Staubli VAL3: refreshImport.pgx

program refreshImport(bool x_bShowLine (dimensions=1), string& x_sPath[] (dimensions=1))
  local num l_nLocal
  local string l_sEmpty
  local string l_sItem
begin
  //
  call use2:setSizeList(0,0,17,11)
  call use2:listcreate("USB")
  call use:stringCopy(l_sEmpty,sImport)
  call use2:listempty()
  //
  // build the list
  if libList(x_sPath[1],sImport)
    // build and refresh
    if x_sPath[1]!="USB0://"
      l_sItem=".."
      call use2:listadd(l_sItem)
    endIf
    call use2:listadd(sImport)
    use2:nView=nViewImport
    call use2:listredraw(nIndexImport-nViewImport)
    if !x_bShowLine
      call use2:listcursor(nViewImport,false)
    endIf
  endIf
end
